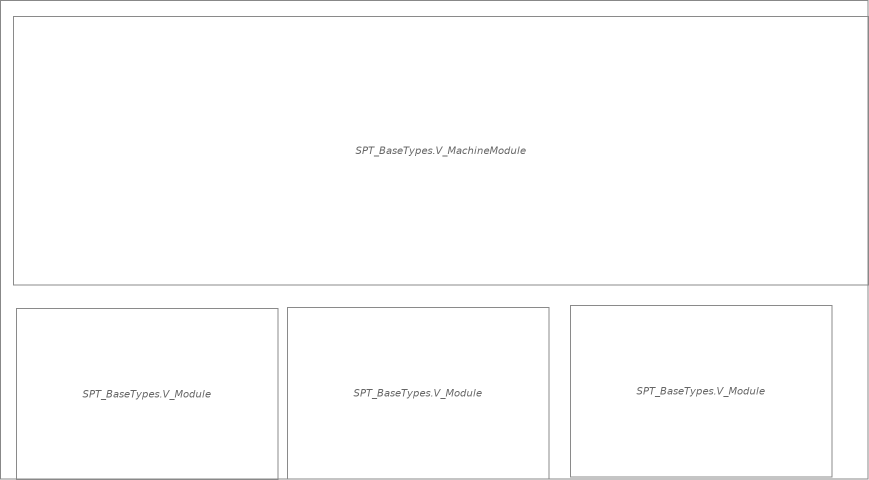
VISUALIZATION Visualization  // 869x480
    Frame (13,16 856x269)
        shows SPT_BaseTypes.V_MachineModule(HMI := MAIN.Machine.PackMLBaseModule_HMI)
    Frame (16,308 262x172)
        shows SPT_BaseTypes.V_Module(HMI := MAIN.Machine.Draw.PackMLBaseModule_HMI)
    Frame (287,307 262x172)
        shows SPT_BaseTypes.V_Module(HMI := MAIN.Machine.Unwind.PackMLBaseModule_HMI)
    Frame (570,305 262x172)
        shows SPT_BaseTypes.V_Module(HMI := MAIN.Machine.VirtualMaster.PackMLBaseModule_HMI)
END_VISUALIZATION

(* stored: Version 1.1.0.1, ProductVersion 3.1.4026.12
   Visu Visualization: Id {f14bd933-1c2e-4292-a0e8-45c8972201c4} *)
